PROGRAM MAIN
VAR
END_VAR

END_PROGRAM

(* stored: Version 1.1.0.1
   POU MAIN: Id {4b27a5e2-9aec-49d3-a7c3-49f29d3cbb55} *)
